{attribute 'GeneratedUsingTerminal: EL2521-0124-0016'}
{attribute addProperty BoxType "EL2521-0124-0016"}
{attribute addProperty Id "PLS_EnabledAT %I*BOOL1Status_of_outputAT %I*BOOL1Sync_ErrorAT %I*BOOL1TxPDO_ToggleAT %I*BOOL1"}
{attribute addProperty CRC "2786019635"}
{attribute addProperty Size "4"}
TYPE PLS_Status_A60F4933 :
STRUCT
	{attribute addProperty Name "PLS_Enabled"}
	PLS_Enabled AT %I* : BOOL;
	{attribute addProperty Name "Status_of_output"}
	Status_of_output AT %I* : BOOL;
	{attribute addProperty Name "Sync_Error"}
	Sync_Error AT %I* : BOOL;
	{attribute addProperty Name "TxPDO_Toggle"}
	TxPDO_Toggle AT %I* : BOOL;
END_STRUCT
END_TYPE

(* stored: Version 1.2.0.0, ProductVersion 3.1.4024.9
   DUT PLS_Status_A60F4933: Id {4e386fd3-1fa6-4c9d-893f-bea080ade6b2} *)
